FUNCTION F_NOW (* returns current local date and time *)
  (* Standard: 61499-1; Description: Copyright (c) 2024 HR Agrartechnik GmbH This program and the accompanying materials are made available under the terms of the Eclipse Public License 2.0 which is available at https://www.eclipse.org/legal/epl-2.0/ SPDX-License-Identifier: EPL-2.0 returns current local date and time This may be affect to step changes (e.g., adjusting winter/summer time). (This is only a Wrapper around the ST Function NOW) *)
  (* Version 3.0, 2025-04-14, Patrick Aigner, changed package *)
  (* Version 1.0, 2024-10-01, Franz Höpfinger, HR Agrartechnik GmbH *)
  PACKAGE utils::timing;
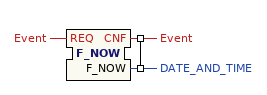
  EVENT_INPUT
    REQ;
  END_EVENT
  EVENT_OUTPUT
    CNF WITH F_NOW;
  END_EVENT
  VAR_OUTPUT
    F_NOW : DATE_AND_TIME;
  END_VAR
  BODY IN ST:
PACKAGE utils::timing;

(* returns current local date and time *)
FUNCTION F_NOW : DATE_AND_TIME
F_NOW := NOW();
END_FUNCTION
  END_BODY
END_FUNCTION
